PROGRAM INTERNAL MAIN

END_PROGRAM

(* stored: Version 1.1.0.1, ProductVersion 3.1.4024.6
   POU MAIN: Id {c1cce3e1-4613-0251-2ba8-0af5f6aff08c}, SpecialFunc None *)
